{attribute 'qualified_only'}
VAR_GLOBAL
	//units mm
linearpos	:linearPositions;
	//units degrees
	InstrumentPositions	:ARRAY [0..7] OF LREAL	:=[0,60,120,180,240,300,35];

	
END_VAR

(* stored: Version 1.1.0.1, ProductVersion 3.1.4024.12
   GVL MovementPositions: Id {a66a7354-78bb-46fc-84f3-bc173096fb3b} *)
